TYPE ST_Element :
STRUCT
	sName		:STRING;
END_STRUCT
END_TYPE

(* stored: Version 1.1.0.1
   DUT ST_Element: Id {d8eccb6c-81c3-498d-b1c6-4d94b9a98778} *)
